(* CODESYS project tcunits.library
   Author: Roald Ruiter
   Placeholder: TcUnits
   Title: TcUnits
   Version: 0.1.0
   Description: Aliases for units
   Company: Roald

Project tree, tasks and I/O mapping:
  Distance/
    data type Millimeter
  Force/
    data type Newton
  Speed/
    data type MillimeterPerSecond
  Time/
    data type Millisecond
  Torque/
    data type NewtonMeter
  Weight/
    data type Kilogram
  data type Percent
*)

// Distance/Millimeter
TYPE Millimeter : LREAL;
END_TYPE

// Force/Newton
TYPE Newton : LREAL;
END_TYPE

// Speed/MillimeterPerSecond
TYPE MillimeterPerSecond : LREAL;
END_TYPE

// Time/Millisecond
TYPE Millisecond : LREAL;
END_TYPE

// Torque/NewtonMeter
TYPE NewtonMeter : LREAL;
END_TYPE

// Weight/Kilogram
TYPE Kilogram : LREAL;
END_TYPE

// Percent
TYPE Percent : LREAL;
END_TYPE
